KUKA KRL program: ps_res_c1.src, ps_res_c1.dat

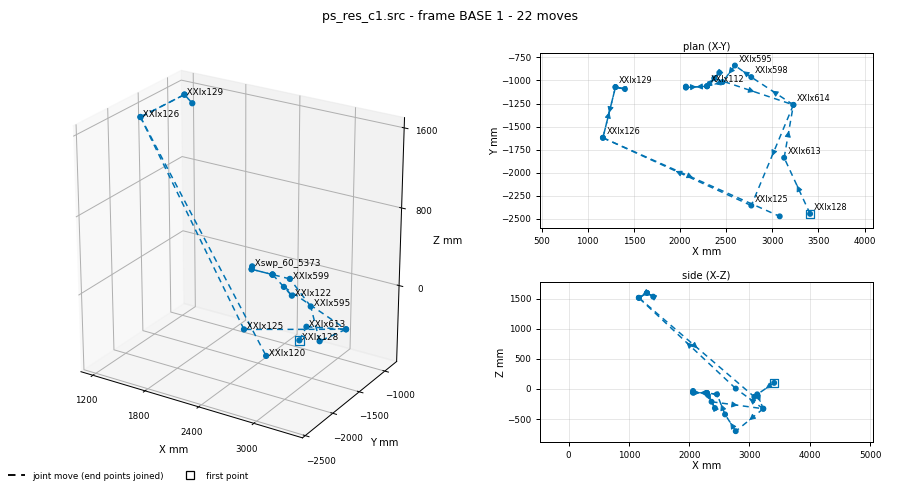
[picture p0: tool path of ps_res_c1.src in frame BASE 1, 22 of 22 moves have a stored position in this frame; points joined in program order, loops and branches not executed]
--- ps_res_c1.src ---
&ACCESS RVO
&REL 5
&COMMENT Solda GUN C1 respot
&PARAM DISKPATH = KRC:\R1\Program
DEF ps_res_c1( )

;FOLD INI
;FOLD SPOTTECH INI
USERSPOT(#INIT)
;ENDFOLD (SPOTTECH INI)
;FOLD GRIPPERTECH INI
USER_GRP(0,DUMMY,DUMMY,GDEFAULT)
;ENDFOLD (GRIPPERTECH INI)
  ;FOLD USER INI
    ;Make your modifications here

  ;ENDFOLD (USER INI)
;ENDFOLD (INI)

; Caracterização dos meios de produção:
; Versão Atual:
; 08/06/2013 12:00 Name: P13.050-R1 CHANGES: Solda respot Actros
; Gun C1 (F2 6640 0018 984)

chk_w2_wechs_ok ( )              ; CHECK C1

if MaxStandMenge (1) then
 MaxStandmengeErreicht (1)
endif

IF (NOT(GHOST())) THEN
if Elektrodenwechsel (1) then
 e_fraes2 ()
endif
ENDIF

;FOLD PTP Xlx128 CONT Vel=100 % PDAT35 Tool[2]:GUN C1 Base[1]:Actros;%{PE}%R 8.2.20,%MKUKATPBASIS,%CMOVE,%VPTP,%P 1:PTP, 2:Xlx128, 3:C_DIS, 5:100, 7:PDAT35
$BWDSTART=FALSE
PDAT_ACT=PPDAT35
FDAT_ACT=FXlx128
BAS(#PTP_PARAMS,100)
PTP XXlx128 C_DIS
;ENDFOLD

;FOLD OUT 3334 'R1 solicita lib. soldar respot' State=TRUE ;%{PE}%R 8.2.20,%MKUKATPBASIS,%COUT,%VOUTX,%P 2:3334, 3:R1 solicita lib. soldar respot, 5:TRUE, 6:
$OUT[3334]=TRUE
;ENDFOLD
;FOLD WAIT FOR ( IN 3334 'Aguarda lib. Soldar respot' );%{PE}%R 8.2.20,%MKUKATPBASIS,%CEXT_WAIT_FOR,%VEXT_WAIT_FOR,%P 2:, 4:, 5:$IN, 6:3334, 7:Aguarda lib. Soldar respot, 9:
WAIT FOR  ( $IN[3334] )
;ENDFOLD
;FOLD OUT 3334 'R1 solicita lib. soldar respot' State=FALSE ;%{PE}%R 8.2.20,%MKUKATPBASIS,%COUT,%VOUTX,%P 2:3334, 3:R1 solicita lib. soldar respot, 5:FALSE, 6:
$OUT[3334]=FALSE
;ENDFOLD

;FOLD PTP Xlx613 CONT Vel=100 % PDAT9 Tool[2]:GUN C1 Base[1]:Actros;%{PE}%R 8.2.19,%MKUKATPBASIS,%CMOVE,%VPTP,%P 1:PTP, 2:Xlx613, 3:C_DIS, 5:100, 7:PDAT9
$BWDSTART=FALSE
PDAT_ACT=PPDAT9
FDAT_ACT=FXlx613
BAS(#PTP_PARAMS,100)
PTP XXlx613 C_DIS
;ENDFOLD
;FOLD PTP Xlx614 CONT Vel=100 % PDAT10 Tool[2]:GUN C1 Base[1]:Actros;%{PE}%R 8.2.19,%MKUKATPBASIS,%CMOVE,%VPTP,%P 1:PTP, 2:Xlx614, 3:C_DIS, 5:100, 7:PDAT10
$BWDSTART=FALSE
PDAT_ACT=PPDAT10
FDAT_ACT=FXlx614
BAS(#PTP_PARAMS,100)
PTP XXlx614 C_DIS
;ENDFOLD
;FOLD PTP Xlx598 CONT Vel=100 % PDAT12 Tool[2]:GUN C1 Base[1]:Actros;%{PE}%R 8.2.19,%MKUKATPBASIS,%CMOVE,%VPTP,%P 1:PTP, 2:Xlx598, 3:C_DIS, 5:100, 7:PDAT12
$BWDSTART=FALSE
PDAT_ACT=PPDAT12
FDAT_ACT=FXlx598
BAS(#PTP_PARAMS,100)
PTP XXlx598 C_DIS
;ENDFOLD
;FOLD PTP Xlx595 CONT Vel=100 % PDAT13 Tool[2]:GUN C1 Base[1]:Actros;%{PE}%R 8.2.19,%MKUKATPBASIS,%CMOVE,%VPTP,%P 1:PTP, 2:Xlx595, 3:C_DIS, 5:100, 7:PDAT13
$BWDSTART=FALSE
PDAT_ACT=PPDAT13
FDAT_ACT=FXlx595
BAS(#PTP_PARAMS,100)
PTP XXlx595 C_DIS
;ENDFOLD
;FOLD PTP Xlx599 CONT Vel=100 % PDAT14 Tool[2]:GUN C1 Base[1]:Actros;%{PE}%R 8.2.19,%MKUKATPBASIS,%CMOVE,%VPTP,%P 1:PTP, 2:Xlx599, 3:C_DIS, 5:100, 7:PDAT14
$BWDSTART=FALSE
PDAT_ACT=PPDAT14
FDAT_ACT=FXlx599
BAS(#PTP_PARAMS,100)
PTP XXlx599 C_DIS
;ENDFOLD
;FOLD PTP Xlx112 CONT Vel=100 % PDAT16 Tool[2]:GUN C1 Base[1]:Actros;%{PE}%R 8.2.19,%MKUKATPBASIS,%CMOVE,%VPTP,%P 1:PTP, 2:Xlx112, 3:C_DIS, 5:100, 7:PDAT16
$BWDSTART=FALSE
PDAT_ACT=PPDAT16
FDAT_ACT=FXlx112
BAS(#PTP_PARAMS,100)
PTP XXlx112 C_DIS
;ENDFOLD
;FOLD PTP Xlx111 CONT Vel=100 % PDAT15 Tool[2]:GUN C1 Base[1]:Actros;%{PE}%R 8.2.19,%MKUKATPBASIS,%CMOVE,%VPTP,%P 1:PTP, 2:Xlx111, 3:C_DIS, 5:100, 7:PDAT15
$BWDSTART=FALSE
PDAT_ACT=PPDAT15
FDAT_ACT=FXlx111
BAS(#PTP_PARAMS,100)
PTP XXlx111 C_DIS
;ENDFOLD

;FOLD ; swp_60_5373;%{PE}%R 8.2.20,%MKUKATPBASIS,%CCOMMENT,%VNORMAL,%P 2:swp_60_5373
;ENDFOLD
;FOLD PTP swp_60_5373 P_OLP7 SPOT Gun=1 RETR OPN PgNo1=47 ACTIVE=1 Tool[2]:GUN C1 Base[1]:Actros;%{PE}%R 8.2.2,%MKUKATPSPOT,%CSPOT,%VPTP,%P 1:PTP, 2:swp_60_5373, 3:, 5:100, 7:P_OLP7, 10:1, 12:#FIRST, 14:#OPN, 16:47, 18:1, 20:1, 22:0, 24:1, 25:S_OLP1
$BWDSTART=FALSE
PDAT_ACT=PP_OLP7
FDAT_ACT=Fswp_60_5373
BAS(#PTP_PARAMS,PP_OLP7.VEL)
S_ACT.GUN=1
S_ACT.PAIR=SDEFAULT.PAIR
S_ACT.RETR=#OPN
S_ACT.CLO_TM=1
S_ACT.PGNO1=47
S_ACT.PGNO2=SDEFAULT.PGNO2
S_ACT.PRESS1=SDEFAULT.PRESS1
S_ACT.PRESS2=SDEFAULT.PRESS2
S_READY=FALSE
PTP Xswp_60_5373
USERSPOT(#SPOT, S_ACT)
WAIT FOR S_READY
;ENDFOLD

;FOLD PTP Xlx114 CONT Vel=100 % PDAT18 Tool[2]:GUN C1 Base[1]:Actros;%{PE}%R 8.2.19,%MKUKATPBASIS,%CMOVE,%VPTP,%P 1:PTP, 2:Xlx114, 3:C_DIS, 5:100, 7:PDAT18
$BWDSTART=FALSE
PDAT_ACT=PPDAT18
FDAT_ACT=FXlx114
BAS(#PTP_PARAMS,100)
PTP XXlx114 C_DIS
;ENDFOLD
;FOLD PTP Xlx113 CONT Vel=100 % PDAT17 Tool[2]:GUN C1 Base[1]:Actros;%{PE}%R 8.2.19,%MKUKATPBASIS,%CMOVE,%VPTP,%P 1:PTP, 2:Xlx113, 3:C_DIS, 5:100, 7:PDAT17
$BWDSTART=FALSE
PDAT_ACT=PPDAT17
FDAT_ACT=FXlx113
BAS(#PTP_PARAMS,100)
PTP XXlx113 C_DIS
;ENDFOLD
;FOLD PTP Xlx214 CONT Vel=100 % P_OLP8 Tool[2]:GUN C1 Base[1]:Actros;%{PE}%R 8.2.19,%MKUKATPBASIS,%CMOVE,%VPTP,%P 1:PTP, 2:Xlx214, 3:C_DIS, 5:100, 7:P_OLP8
$BWDSTART=FALSE
PDAT_ACT=PP_OLP8
FDAT_ACT=FXlx214
BAS(#PTP_PARAMS,100)
PTP XXlx214 C_DIS
;ENDFOLD
;FOLD PTP Xlx122 CONT Vel=100 % PDAT28 Tool[2]:GUN C1 Base[1]:Actros;%{PE}%R 8.2.19,%MKUKATPBASIS,%CMOVE,%VPTP,%P 1:PTP, 2:Xlx122, 3:C_DIS, 5:100, 7:PDAT28
$BWDSTART=FALSE
PDAT_ACT=PPDAT28
FDAT_ACT=FXlx122
BAS(#PTP_PARAMS,100)
PTP XXlx122 C_DIS
;ENDFOLD
;FOLD PTP Xlx116 CONT Vel=100 % PDAT20 Tool[2]:GUN C1 Base[1]:Actros;%{PE}%R 8.2.19,%MKUKATPBASIS,%CMOVE,%VPTP,%P 1:PTP, 2:Xlx116, 3:C_DIS, 5:100, 7:PDAT20
$BWDSTART=FALSE
PDAT_ACT=PPDAT20
FDAT_ACT=FXlx116
BAS(#PTP_PARAMS,100)
PTP XXlx116 C_DIS
;ENDFOLD
;FOLD PTP Xlx118 CONT Vel=100 % PDAT22 Tool[2]:GUN C1 Base[1]:Actros;%{PE}%R 8.2.19,%MKUKATPBASIS,%CMOVE,%VPTP,%P 1:PTP, 2:Xlx118, 3:C_DIS, 5:100, 7:PDAT22
$BWDSTART=FALSE
PDAT_ACT=PPDAT22
FDAT_ACT=FXlx118
BAS(#PTP_PARAMS,100)
PTP XXlx118 C_DIS
;ENDFOLD
;FOLD PTP Xlx125 CONT Vel=100 % PDAT32 Tool[2]:GUN C1 Base[1]:Actros;%{PE}%R 8.2.20,%MKUKATPBASIS,%CMOVE,%VPTP,%P 1:PTP, 2:Xlx125, 3:C_DIS, 5:100, 7:PDAT32
$BWDSTART=FALSE
PDAT_ACT=PPDAT32
FDAT_ACT=FXlx125
BAS(#PTP_PARAMS,100)
PTP XXlx125 C_DIS
;ENDFOLD

;FOLD Collision.Monitoring_3_On ;%{PE}%MKUKATPUSER
COLLSTOP( 3, 1 ) ;Interrupt-Controlled
;ENDFOLD

;FOLD PTP Xlx126 CONT Vel=100 % PDAT33 Tool[2]:GUN C1 Base[1]:Actros;%{PE}%R 8.2.20,%MKUKATPBASIS,%CMOVE,%VPTP,%P 1:PTP, 2:Xlx126, 3:C_DIS, 5:100, 7:PDAT33
$BWDSTART=FALSE
PDAT_ACT=PPDAT33
FDAT_ACT=FXlx126
BAS(#PTP_PARAMS,100)
PTP XXlx126 C_DIS
;ENDFOLD

;FOLD Collision.Monitoring_5_On ;%{PE}%MKUKATPUSER
COLLSTOP( 5, 1 ) ;not Interrupt-Controlled
;ENDFOLD

;FOLD PTP Xlx129 CONT Vel=100 % PDAT30 Tool[2]:GUN C1 Base[1]:Actros;%{PE}%R 8.2.20,%MKUKATPBASIS,%CMOVE,%VPTP,%P 1:PTP, 2:Xlx129, 3:C_DIS, 5:100, 7:PDAT30
$BWDSTART=FALSE
PDAT_ACT=PPDAT30
FDAT_ACT=FXlx129
BAS(#PTP_PARAMS,100)
PTP XXlx129 C_DIS
;ENDFOLD

;FOLD ; swp_60_5655;%{PE}%R 8.2.20,%MKUKATPBASIS,%CCOMMENT,%VNORMAL,%P 2:swp_60_5655
;ENDFOLD
;FOLD PTP swp_60_5656 P_OLP23 SPOT Gun=1 RETR OPN PgNo1=48 ACTIVE=1 Tool[2]:GUN C1 Base[1]:Actros;%{PE}%R 8.2.2,%MKUKATPSPOT,%CSPOT,%VPTP,%P 1:PTP, 2:swp_60_5656, 3:, 5:100, 7:P_OLP23, 10:1, 12:#FIRST, 14:#OPN, 16:48, 18:1, 20:1, 22:0, 24:1, 25:S_OLP2
$BWDSTART=FALSE
PDAT_ACT=PP_OLP23
FDAT_ACT=Fswp_60_5656
BAS(#PTP_PARAMS,PP_OLP23.VEL)
S_ACT.GUN=1
S_ACT.PAIR=SDEFAULT.PAIR
S_ACT.RETR=#OPN
S_ACT.CLO_TM=1
S_ACT.PGNO1=48
S_ACT.PGNO2=SDEFAULT.PGNO2
S_ACT.PRESS1=SDEFAULT.PRESS1
S_ACT.PRESS2=SDEFAULT.PRESS2
S_READY=FALSE
PTP Xswp_60_5656
USERSPOT(#SPOT, S_ACT)
WAIT FOR S_READY
;ENDFOLD

;FOLD PTP Xlx130 CONT Vel=100 % PDAT31 Tool[2]:GUN C1 Base[1]:Actros;%{PE}%R 8.2.20,%MKUKATPBASIS,%CMOVE,%VPTP,%P 1:PTP, 2:Xlx130, 3:C_DIS, 5:100, 7:PDAT31
$BWDSTART=FALSE
PDAT_ACT=PPDAT31
FDAT_ACT=FXlx130
BAS(#PTP_PARAMS,100)
PTP XXlx130 C_DIS
;ENDFOLD
;FOLD PTP Xlx124 CONT Vel=100 % PDAT29 Tool[2]:GUN C1 Base[1]:Actros;%{PE}%R 8.2.19,%MKUKATPBASIS,%CMOVE,%VPTP,%P 1:PTP, 2:Xlx124, 3:C_DIS, 5:100, 7:PDAT29
$BWDSTART=FALSE
PDAT_ACT=PPDAT29
FDAT_ACT=FXlx124
BAS(#PTP_PARAMS,100)
PTP XXlx124 C_DIS
;ENDFOLD

;FOLD Collision.Monitoring_5_Off . ;%{PE}%MKUKATPUSER
COLLSTOP( 5, 2+0 )
;ENDFOLD

;FOLD PTP Xlx120 CONT Vel=100 % PDAT24 Tool[2]:GUN C1 Base[1]:Actros;%{PE}%R 8.2.19,%MKUKATPBASIS,%CMOVE,%VPTP,%P 1:PTP, 2:Xlx120, 3:C_DIS, 5:100, 7:PDAT24
$BWDSTART=FALSE
PDAT_ACT=PPDAT24
FDAT_ACT=FXlx120
BAS(#PTP_PARAMS,100)
PTP XXlx120 C_DIS
;ENDFOLD

;FOLD Collision.Monitoring_3_Off . ;%{PE}%MKUKATPUSER
COLLSTOP( 3, 2+0 )
;ENDFOLD

IF (NOT(GHOST())) THEN
if FraesAnf (1) then
 f_fraes2 ()
endif
ENDIF
END

--- ps_res_c1.dat ---
&ACCESS RVO
&REL 5
&COMMENT Solda GUN C1 respot
&PARAM DISKPATH = KRC:\R1\Program
DEFDAT ps_res_c1
;FOLD EXTERNAL DECLARATIONS;%{PE}%MKUKATPBASIS,%CEXT,%VCOMMON,%P
;FOLD GRIPPERTECH EXT
EXT  H50 (INT  :IN,INT  :IN,INT  :IN,GRP_TYP  :IN )
;ENDFOLD (GRIPPERTECH EXT)
;FOLD SPOTTECH EXT
EXT  USERSPOT (S_COMMAND  :IN,SPOT_TYPE  :IN )
;ENDFOLD (SPOTTECH EXT)
;FOLD BASISTECH EXT;%{PE}%MKUKATPBASIS,%CEXT,%VEXT,%P
EXT  BAS (BAS_COMMAND  :IN,REAL  :IN )
DECL INT SUCCESS
;ENDFOLD (BASISTECH EXT)
;FOLD USER EXT;%{E}%MKUKATPUSER,%CEXT,%VEXT,%P
;Make your modifications here

;ENDFOLD (USER EXT)
;ENDFOLD (EXTERNAL DECLARATIONS)

;# ============ START PATH : swp_p13050r1_l_res_c1 =============
DECL FDAT Fswp_60_5373={TOOL_NO 2,BASE_NO 1,IPO_FRAME #BASE,POINT2[] " "}
DECL PDAT PP_OLP7={VEL 100.0,ACC 100.0,APO_DIST 0.0}
DECL SPOT_TYPE SS_OLP1={GUN 1,PAIR #FIRST,RETR #CLO,CLO_TM 0,PGNO1 1,PRESS1 1.0,PGNO2 0,PRESS2 0.0}
DECL E6POS Xswp_60_5373={X 2064.0791,Y -1066.35596,Z -32.4513817,A 91.1180573,B -82.0530319,C 89.0981064,S 2,T 42,E1 -4796.72803,E2 0.0,E3 0.0,E4 0.0,E5 0.0,E6 0.0}
DECL PDAT PP_OLP8={VEL 100.0,ACC 100.0,APO_DIST 100.0,APO_MODE #CDIS}
DECL SPOT_TYPE SS_OLP2={GUN 1,PAIR #FIRST,RETR #CLO,CLO_TM 0,PGNO1 1,PRESS1 1.0,PGNO2 0,PRESS2 0.0}
DECL BASIS_SUGG_T LAST_BASIS={POINT1[] "Xlx131                  ",POINT2[] "Xlx131                  ",CP_PARAMS[] "CPDAT0                  ",PTP_PARAMS[] "PDAT36                  ",CONT[] "C_DIS                   ",CP_VEL[] "2.0                     ",PTP_VEL[] "100                     ",SYNC_PARAMS[] "SYNCDAT                 ",SPL_NAME[] "S0                      "}
DECL PDAT PPDAT9={VEL 100.0,ACC 100.0,APO_DIST 100.0,APO_MODE #CDIS}
DECL E6POS XXlx613={X 3128.59912,Y -1837.60901,Z -88.7565308,A -40.3791695,B 5.19717216,C -2.13011694,S 2,T 10,E1 -3882.32593,E2 0.0,E3 0.0,E4 0.0,E5 0.0,E6 0.0}
DECL FDAT FXlx613={TOOL_NO 2,BASE_NO 1,IPO_FRAME #BASE,POINT2[] " ",TQ_STATE FALSE}
DECL PDAT PPDAT10={VEL 100.0,ACC 100.0,APO_DIST 100.0,APO_MODE #CDIS}
DECL E6POS XXlx614={X 3228.57397,Y -1264.50903,Z -327.245514,A -61.542881,B 4.42272997,C -3.29499197,S 2,T 10,E1 -3896.23511,E2 0.0,E3 0.0,E4 0.0,E5 0.0,E6 0.0}
DECL FDAT FXlx614={TOOL_NO 2,BASE_NO 1,IPO_FRAME #BASE,POINT2[] " ",TQ_STATE FALSE}
DECL PDAT PPDAT12={VEL 100.0,ACC 100.0,APO_DIST 100.0,APO_MODE #CDIS}
DECL E6POS XXlx598={X 2772.13696,Y -963.370972,Z -700.090515,A -108.568497,B -22.3504105,C -31.4689198,S 2,T 10,E1 -4756.625,E2 0.0,E3 0.0,E4 0.0,E5 0.0,E6 0.0}
DECL FDAT FXlx598={TOOL_NO 2,BASE_NO 1,IPO_FRAME #BASE,POINT2[] " ",TQ_STATE FALSE}
DECL PDAT PPDAT13={VEL 100.0,ACC 100.0,APO_DIST 100.0,APO_MODE #CDIS}
DECL E6POS XXlx595={X 2595.06812,Y -838.345276,Z -421.61911,A -115.791,B -50.3485718,C -66.9213181,S 2,T 10,E1 -5055.82715,E2 0.0,E3 0.0,E4 0.0,E5 0.0,E6 0.0}
DECL FDAT FXlx595={TOOL_NO 2,BASE_NO 1,IPO_FRAME #BASE,POINT2[] " ",TQ_STATE FALSE}
DECL PDAT PPDAT14={VEL 100.0,ACC 100.0,APO_DIST 100.0,APO_MODE #CDIS}
DECL E6POS XXlx599={X 2461.47095,Y -1017.10797,Z -88.183609,A -90.2153397,B -44.6350708,C -89.307579,S 2,T 10,E1 -4661.64697,E2 0.0,E3 0.0,E4 0.0,E5 0.0,E6 0.0}
DECL FDAT FXlx599={TOOL_NO 2,BASE_NO 1,IPO_FRAME #BASE,POINT2[] " ",TQ_STATE FALSE}
DECL E6POS XXLX111={X 2064.1731,Y -1075.797,Z -59.6603317,A 91.1172333,B -82.0564575,C 89.0994492,S 2,T 42,E1 -4796.72803,E2 0.0,E3 0.0,E4 0.0,E5 0.0,E6 0.0}
DECL FDAT FXlx111={TOOL_NO 2,BASE_NO 1,IPO_FRAME #BASE,POINT2[] " ",TQ_STATE FALSE}
DECL PDAT PPDAT15={VEL 100.0,ACC 100.0,APO_DIST 100.0,APO_MODE #CDIS}
DECL E6POS XXLX112={X 2293.125,Y -1062.66003,Z -65.5999527,A 92.1322403,B -86.1724472,C 88.0859528,S 2,T 42,E1 -4796.72803,E2 0.0,E3 0.0,E4 0.0,E5 0.0,E6 0.0}
DECL FDAT FXlx112={TOOL_NO 2,BASE_NO 1,IPO_FRAME #BASE,POINT2[] " ",TQ_STATE FALSE}
DECL PDAT PPDAT16={VEL 100.0,ACC 100.0,APO_DIST 100.0,APO_MODE #CDIS}
DECL E6POS XXLX113={X 2293.09204,Y -1062.47595,Z -65.7701492,A 92.2209091,B -86.1646576,C 87.9893265,S 2,T 42,E1 -4796.72607,E2 0.0,E3 0.0,E4 0.0,E5 0.0,E6 0.0}
DECL FDAT FXlx113={TOOL_NO 2,BASE_NO 1,IPO_FRAME #BASE,POINT2[] " ",TQ_STATE FALSE}
DECL PDAT PPDAT17={VEL 100.0,ACC 100.0,APO_DIST 100.0,APO_MODE #CDIS}
DECL E6POS XXLX114={X 2064.15601,Y -1075.771,Z -59.5123482,A 91.0795822,B -82.0516129,C 89.1374588,S 2,T 42,E1 -4796.729,E2 0.0,E3 0.0,E4 0.0,E5 0.0,E6 0.0}
DECL FDAT FXlx114={TOOL_NO 2,BASE_NO 1,IPO_FRAME #BASE,POINT2[] " ",TQ_STATE FALSE}
DECL PDAT PPDAT18={VEL 100.0,ACC 100.0,APO_DIST 100.0,APO_MODE #CDIS}
DECL E6POS XXLX214={X 2293.13599,Y -1062.69397,Z -65.5598679,A 92.1095428,B -86.1729279,C 88.109993,S 2,T 42,E1 -4796.72705,E2 0.0,E3 0.0,E4 0.0,E5 0.0,E6 0.0}
DECL FDAT FXlx214={TOOL_NO 2,BASE_NO 1,IPO_FRAME #BASE,POINT2[] " ",TQ_STATE FALSE}
DECL E6POS XXLX116={X 2371.28589,Y -976.845276,Z -211.696899,A -173.527893,B -42.2611313,C -21.4320107,S 2,T 42,E1 -4744.07617,E2 0.0,E3 0.0,E4 0.0,E5 0.0,E6 0.0}
DECL FDAT FXlx116={TOOL_NO 2,BASE_NO 1,IPO_FRAME #BASE,POINT2[] " ",TQ_STATE FALSE}
DECL PDAT PPDAT20={VEL 100.0,ACC 100.0,APO_DIST 100.0,APO_MODE #CDIS}
DECL E6POS XXLX118={X 3228.51001,Y -1264.5,Z -327.250488,A -61.5434799,B 4.42404079,C -3.29771996,S 2,T 10,E1 -3896.23511,E2 0.0,E3 0.0,E4 0.0,E5 0.0,E6 0.0}
DECL FDAT FXlx118={TOOL_NO 2,BASE_NO 1,IPO_FRAME #BASE,POINT2[] " ",TQ_STATE FALSE}
DECL PDAT PPDAT22={VEL 100.0,ACC 100.0,APO_DIST 100.0,APO_MODE #CDIS}
DECL E6POS XXLX120={X 3080.58911,Y -2472.3811,Z -130.077301,A -5.5123291,B 6.21072912,C -0.00073081709,S 2,T 10,E1 -3859.23389,E2 0.0,E3 0.0,E4 0.0,E5 0.0,E6 0.0}
DECL FDAT FXlx120={TOOL_NO 2,BASE_NO 1,IPO_FRAME #BASE,POINT2[] " ",TQ_STATE FALSE}
DECL PDAT PPDAT24={VEL 100.0,ACC 100.0,APO_DIST 100.0,APO_MODE #CDIS}
DECL E6POS XXLX122={X 2426.23389,Y -916.041016,Z -316.144897,A -176.385696,B -55.5256882,C -4.98000813,S 2,T 42,E1 -4763.18506,E2 0.0,E3 0.0,E4 0.0,E5 0.0,E6 0.0}
DECL FDAT FXlx122={TOOL_NO 2,BASE_NO 1,IPO_FRAME #BASE,POINT2[] " ",TQ_STATE FALSE}
DECL PDAT PPDAT28={VEL 100.0,ACC 100.0,APO_DIST 100.0,APO_MODE #CDIS}
DECL E6POS XXLX124={X 1164.94495,Y -1621.10706,Z 1512.08997,A 10.60044,B 58.1972809,C 68.5988312,S 2,T 34,E1 -5491.97705,E2 0.0,E3 0.0,E4 0.0,E5 0.0,E6 0.0}
DECL FDAT FXlx124={TOOL_NO 2,BASE_NO 1,IPO_FRAME #BASE,POINT2[] " ",TQ_STATE FALSE}
DECL PDAT PPDAT29={VEL 100.0,ACC 100.0,APO_DIST 100.0,APO_MODE #CDIS}
DECL SPOT_SUGG_T LAST_SPOT={GUN[] "1                       ",RETR_CMD[] "#OPN                    ",CHOISE[] "#FIRST                  ",CLO_TM[] "0                       ",PGNO1[] "1                       ",PRESS1[] "0                       ",PGNO2[] "1                       ",PRESS2[] "0                       ",SPOT_PARAMS[] "NORMAL                  "}
DECL PDAT PPDAT30={VEL 100.0,ACC 100.0,APO_DIST 100.0,APO_MODE #CDIS}
DECL E6POS XXlx129={X 1301.15601,Y -1072.01099,Z 1592.88599,A 0.915633321,B 44.6264191,C 90.567688,S 2,T 34,E1 -5823.46582,E2 0.0,E3 0.0,E4 0.0,E5 0.0,E6 0.0}
DECL FDAT FXlx129={TOOL_NO 2,BASE_NO 1,IPO_FRAME #BASE,POINT2[] " ",TQ_STATE FALSE}
DECL PDAT PP_OLP23={VEL 100.0,ACC 100.0,APO_DIST 0.0}
DECL E6POS Xswp_60_5656={X 1403.47705,Y -1092.578,Z 1531.23901,A 0.986616373,B 44.6927681,C 90.6115494,S 2,T 34,E1 -5823.46387,E2 0.0,E3 0.0,E4 0.0,E5 0.0,E6 0.0}
DECL FDAT Fswp_60_5656={TOOL_NO 2,BASE_NO 1,IPO_FRAME #BASE,POINT2[] " ",TQ_STATE FALSE}
DECL PDAT PPDAT31={VEL 100.0,ACC 100.0,APO_DIST 100.0,APO_MODE #CDIS}
DECL E6POS XXlx130={X 1301.15601,Y -1072.01099,Z 1592.88599,A 0.915632427,B 44.6264191,C 90.567688,S 2,T 34,E1 -5823.46582,E2 0.0,E3 0.0,E4 0.0,E5 0.0,E6 0.0}
DECL FDAT FXlx130={TOOL_NO 2,BASE_NO 1,IPO_FRAME #BASE,POINT2[] " ",TQ_STATE FALSE}
DECL E6POS XXLX125={X 2772.58301,Y -2355.36401,Z 6.7653532,A -11.3524399,B 1.41991496,C 11.8210402,S 2,T 2,E1 -4232.19678,E2 0.0,E3 0.0,E4 0.0,E5 0.0,E6 0.0}
DECL FDAT FXlx125={TOOL_NO 2,BASE_NO 1,IPO_FRAME #BASE,POINT2[] " ",TQ_STATE FALSE}
DECL PDAT PPDAT32={VEL 100.0,ACC 100.0,APO_DIST 100.0,APO_MODE #CDIS}
DECL E6POS XXLX126={X 1164.94495,Y -1621.10706,Z 1512.08997,A 10.60044,B 58.1972809,C 68.5988312,S 2,T 34,E1 -5491.97705,E2 0.0,E3 0.0,E4 0.0,E5 0.0,E6 0.0}
DECL FDAT FXlx126={TOOL_NO 2,BASE_NO 1,IPO_FRAME #BASE,POINT2[] " ",TQ_STATE FALSE}
DECL PDAT PPDAT33={VEL 100.0,ACC 100.0,APO_DIST 100.0,APO_MODE #CDIS}
DECL E6POS XXLX128={X 3409.55396,Y -2445.41211,Z 101.452698,A 10.5908098,B 25.0753708,C 8.57575226,S 2,T 2,E1 -2854.21997,E2 0.0,E3 0.0,E4 0.0,E5 0.0,E6 0.0}
DECL FDAT FXlx128={TOOL_NO 2,BASE_NO 1,IPO_FRAME #BASE,POINT2[] " ",TQ_STATE FALSE}
DECL PDAT PPDAT35={VEL 100.0,ACC 100.0,APO_DIST 100.0,APO_MODE #CDIS}
ENDDAT
